INTERFACE PUBLIC AbortedCommands

METHOD PUBLIC Clear
END_METHOD

END_INTERFACE

(* stored: Version 1.1.0.1, ProductVersion 3.1.4026.12
   Itf AbortedCommands: Id {b555524d-549b-0d83-1524-b3f90d512aa1}
   Method Clear: Id {9c2659ef-9635-02bc-21a0-221ddb076b01} *)
